# B&R Automation Studio project LW1
Automation Studio 4.9

## Configuration Config1

CPU 4PP065.0571-P74, AutomationRuntime D4.63, Build 4.1.2, Vc V4.73.2

### Task classes (Cpu.sw)
```
Cyclic#4:
  Program <- Program.prg
Binaries: udbdef, FWRules, TCData, sysconf, Role, User, iomap, ashwd, asfw, arconfig, ashwac
Libraries: MotorCtrl
```

### Hardware
```
4PP065_0571_P74 : 4PP065.0571-P74 v1.2.0.0
  Connector IF5:
    ActivateDevice = 1
  ConfigurationID = ProgSysLab1_Config1
  Simulation = 1
  Cyclic1Duration = 2000
  Cyclic1Tolerance = 2000
```

## Logical view

Binary libraries used (declarations not repeated): operator, runtime, astime, AsIecCon

### Library Logical/Libraries/MotorCtrl (ANSIC)

#### MotorCtrl.fun - Exported functions and function blocks
```iecst
{REDUND_ERROR} FUNCTION_BLOCK FB_Integrator (*TODO: Add your comment here*) (*$GROUP=User,$CAT=User,$GROUPICON=User.png,$CATICON=User.png*)
	VAR_INPUT
		in : REAL;
	END_VAR
	VAR_OUTPUT
		out : REAL;
	END_VAR
	VAR
		dt : REAL;
	END_VAR
END_FUNCTION_BLOCK

{REDUND_ERROR} FUNCTION_BLOCK FB_Motor (*TODO: Add your comment here*) (*$GROUP=User,$CAT=User,$GROUPICON=User.png,$CATICON=User.png*)
	VAR_INPUT
		u : REAL;
	END_VAR
	VAR_OUTPUT
		w : REAL;
		phi : REAL;
	END_VAR
	VAR
		integrator : FB_Integrator;
		Tm : REAL;
		ke : REAL;
		dt : REAL;
		oldw : REAL;
	END_VAR
END_FUNCTION_BLOCK

{REDUND_ERROR} FUNCTION_BLOCK FB_Regulator (*TODO: Add your comment here*) (*$GROUP=User,$CAT=User,$GROUPICON=User.png,$CATICON=User.png*)
	VAR_INPUT
		e : REAL;
	END_VAR
	VAR_OUTPUT
		u : REAL;
	END_VAR
	VAR
		k_p : REAL;
		k_i : REAL;
		integrator : FB_Integrator;
		iyOld : REAL;
		max_abs_value : REAL;
		dt : REAL;
	END_VAR
END_FUNCTION_BLOCK
```

#### FB_Integrator.c
```c
#include <bur/plctypes.h>
#ifdef __cplusplus
	extern "C"
	{
#endif
	#include "MotorCtrl.h"
#ifdef __cplusplus
	};
#endif
/* TODO: Add your comment here */
void FB_Integrator(struct FB_Integrator* inst)
{
	/*TODO: Add your code here*/
	inst->out = inst->out + inst->in*inst->dt;
}
```

#### FB_Motor.c
```c
#include <bur/plctypes.h>
#ifdef __cplusplus
	extern "C"
	{
#endif
	#include "MotorCtrl.h"
#ifdef __cplusplus
	};
#endif
/* TODO: Add your comment here */
void FB_Motor(struct FB_Motor* inst)
{
	/*TODO: Add your code here*/
	inst->integrator.out = inst->w;
	inst->integrator.in = (inst->u/inst->ke - inst->w) * (inst->dt/inst->Tm);
	FB_Integrator(&inst->integrator);
	inst->integrator.in = inst->w = inst->integrator.out;
	inst->integrator.in *= inst->dt;
	inst->integrator.out = inst->phi;
	FB_Integrator(&inst->integrator);
	inst->phi = inst->integrator.out;
}
```

#### FB_Regulator.c
```c
#include <bur/plctypes.h>
#ifdef __cplusplus
	extern "C"
	{
#endif
	#include "MotorCtrl.h"
#ifdef __cplusplus
	};
#endif
/* TODO: Add your comment here */
void FB_Regulator(struct FB_Regulator* inst)
{
	/*TODO: Add your code here*/
	/*
	inst->integrator.in = inst->e * inst->k_i * inst->dt + inst->iyOld;
	FB_Integrator(&inst->integrator);
	if (inst->e*inst->k_p < inst->max_abs_value)
	{
	inst->iyOld = inst->iyOld - inst->e*inst->k_p - inst->integrator.out;
	if (inst->e*inst->k_p + inst->integrator.out < inst->max_abs_value)
	{
	inst->iyOld = inst->iyOld + inst->e*inst->k_p + inst->integrator.out;
	inst->u = inst->e*inst->k_p + inst->integrator.out;
	}
	else
	{
	inst->iyOld = inst->iyOld + inst->max_abs_value;
	inst->u = inst->max_abs_value;
	}
	}
	else
	{
	inst->iyOld = inst->iyOld - inst->max_abs_value - inst->integrator.out;
	if (inst->max_abs_value + inst->integrator.out < inst->max_abs_value)
	{
	inst->iyOld = inst->iyOld + inst->max_abs_value + inst->integrator.out;
	inst->u = inst->max_abs_value + inst->integrator.out;
	}
	else
	{
	inst->iyOld = inst->iyOld + inst->max_abs_value;
	inst->u = inst->max_abs_value;
	}
	}
	*/

	REAL a = inst->e * inst->k_p;
	REAL b = inst->e * inst->k_i * inst->dt;
	a = a > inst->max_abs_value ? inst->max_abs_value : a;
	a = a < -inst->max_abs_value ? -inst->max_abs_value : a;
	inst->integrator.in = b + inst->iyOld;
	FB_Integrator(&inst->integrator);
	REAL sum = a + inst->integrator.out;
	inst->u = sum;
	inst->u = inst->u > inst->max_abs_value ? inst->max_abs_value : inst->u;
	inst->u = inst->u < -inst->max_abs_value ? -inst->max_abs_value : inst->u;
	inst->iyOld = inst->u - sum;
}
```

### Program Logical/Program

#### Variables.var
```iecst
VAR
	fb_regulator : FB_Regulator;
	fb_motor : FB_Motor;
	fb_motor2 : FB_Motor;
	Speed : REAL;
	Enable : BOOL;
	time : UINT;
END_VAR
```

#### Cyclic.c
```c
#include <bur/plctypes.h>

#ifdef _DEFAULT_INCLUDES
	#include <AsDefault.h>
#endif

void _CYCLIC ProgramCyclic(void)
{
	if (time % 200 == 0)
	{
		Enable = !Enable;

		if (Enable)
		{
			Speed = 100;
		}
		else
		{
			Speed = 0;
		}
	}
	fb_regulator.e = Speed - fb_motor.w;
	FB_Regulator(&fb_regulator);
	fb_motor.u = fb_regulator.u;
	FB_Motor(&fb_motor);
	fb_motor2.u = Speed * fb_motor2.ke;
	FB_Motor(&fb_motor2);

	time += 1;
}
```

#### Init.c
```c
#include <bur/plctypes.h>

#ifdef _DEFAULT_INCLUDES
	#include <AsDefault.h>
#endif

void _INIT ProgramInit(void)
{
	fb_regulator.dt = 0.1;
	fb_regulator.integrator.dt = 0.1;
	fb_regulator.max_abs_value = 24.0;
	fb_regulator.k_p = 0.0064;
	fb_regulator.k_i = 0.16;

	fb_motor.dt = 0.1;
	fb_motor.integrator.dt = 0.1;
	fb_motor.Tm = 0.04;
	fb_motor.ke = 0.048;
	fb_motor.u = 0;

	fb_motor2.dt = 0.1;
	fb_motor2.integrator.dt = 0.1;
	fb_motor2.Tm = 0.04;
	fb_motor2.ke = 0.048;
	fb_motor2.u = 0;

	time = 0;
	Speed = 0;
	Enable = 0;
}
```

Listed in the project but not available here: Logical/Libraries/MotorCtrl/Types.typ, Logical/Libraries/MotorCtrl/Constants.var
